// TIA Portal project "Tesis_taponado" (V20)

(* hardware
DEVICE "S7-1200 station_1"  S7-1200 Station
   slot 0: "Rack_0"  S7-1200 Rack  Rack  V1.0
   slot 1: "PLC_1"  CPU 1214C AC/DC/Rly  6ES7 214-1BG40-0XB0  V4.2
*)

// ===== PLC "PLC_1"  CPU 1214C AC/DC/Rly =====

VAR_GLOBAL   // PLC tag table "Default tag table"
   "I.G" AT %I0.1 : Bool;
   "m" AT %I0.0 : Bool;
   "final_1" AT %I0.6 : Bool;
   "Banda_1" AT %Q0.1 : Bool;
   "E0" AT %M10.0 : Bool;
   "E2" AT %M10.1 : Bool;
   "KT1" AT %M10.2 : Bool;
   "E1" AT %M10.3 : Bool;
   "Fc1" AT %M10.4 : Bool;
   "aux1" AT %M10.5 : Bool;
   "E50" AT %M10.6 : Bool;
   "E51" AT %M10.7 : Bool;
   "E52" AT %M1.0 : Bool;
   "aux2" AT %M11.1 : Bool;
   "final_2" AT %I0.7 : Bool;
   "final_3" AT %I1.0 : Bool;
   "aux3" AT %M11.2 : Bool;
   "final_4" AT %I1.1 : Bool;
   "aux4" AT %M11.3 : Bool;
   "Fc2" AT %M1.4 : Bool;
   "Fc3" AT %M1.5 : Bool;
   "Fc4" AT %M1.6 : Bool;
   "E12" AT %M1.7 : Bool;
   "E92" AT %M2.0 : Bool;
   "E11" AT %M2.1 : Bool;
   "E91" AT %M2.2 : Bool;
   "E10" AT %M2.3 : Bool;
   "E90" AT %M2.4 : Bool;
   "E20" AT %M2.5 : Bool;
   "E32" AT %M2.6 : Bool;
   "E22" AT %M2.7 : Bool;
   "KT2" AT %M3.0 : Bool;
   "E21" AT %M3.1 : Bool;
   "E31" AT %M3.2 : Bool;
   "E30" AT %M3.3 : Bool;
   "E40" AT %M3.4 : Bool;
   "E42" AT %M3.5 : Bool;
   "KT3" AT %M3.6 : Bool;
   "E41" AT %M3.7 : Bool;
   "E72" AT %M4.0 : Bool;
   "E60" AT %M4.1 : Bool;
   "E62" AT %M4.2 : Bool;
   "KT4" AT %M4.3 : Bool;
   "E61" AT %M4.4 : Bool;
   "E71" AT %M4.5 : Bool;
   "E70" AT %M4.6 : Bool;
   "Banda_2" AT %Q0.2 : Bool;
   "Banda_3" AT %Q0.3 : Bool;
   "Banda_4" AT %Q0.0 : Bool;
   "Stopped" AT %M4.7 : Bool;
   "Suspending" AT %I0.2 : Bool;
   "Aborting" AT %I0.3 : Bool;
   "aux5" AT %M5.0 : Bool;
   "UnAbort" AT %M5.1 : Bool;
   "aux6" AT %M5.2 : Bool;
   "Unsuspend" AT %M5.3 : Bool;
   "Starting" AT %M5.4 : Bool;
   "aux7" AT %M5.5 : Bool;
   "aux8" AT %M5.6 : Bool;
   "Starting_Lavado" AT %M5.7 : Bool;
   "aux9" AT %M6.0 : Bool;
   "Starting_Llenado" AT %M6.1 : Bool;
   "aux10" AT %M6.2 : Bool;
   "Starting_Taponado" AT %M6.3 : Bool;
   "aux11" AT %M6.4 : Bool;
   "Starting_Etiquetado" AT %M6.5 : Bool;
   "Start" AT %I0.4 : Bool;
   "Stop_Led" AT %Q0.5 : Bool;
   "Abort_Led" AT %Q1.0 : Bool;
   "Suspend_Led" AT %Q0.7 : Bool;
   "Start_Led" AT %Q1.1 : Bool;
   "aux12" AT %M8.7 : Bool;
END_VAR

DATA_BLOCK "DB1"   // DB1
{ S7_Optimized_Access := 'FALSE' }
VERSION : 0.1
   VAR
      UnAbort : Bool := false;
      Holding_Llenado : Bool;
      Holding_Taponado : Bool;
      Holding_Etiquetado : Bool;
      Holding_Lavado : Bool;
      Completing_Etiquetado : Bool;
      Completing_Taponado : Bool;
      Completing_Llenado : Bool;
      Completing_Lavado : Bool;
      Lavado : Bool;
      Starting : Bool;
      Starting_Lavado : Bool;
      Starting_Llenado : Bool;
      Starting_Taponado : Bool;
      Starting_Etiquetado : Bool;
      Unsuspend : Bool := false;
      Taponado : Bool;
      Etiquetado : Bool;
      Llenado : Bool;
      Aborted : Bool;
      Suspended : Bool;
      starting_plc : Bool;
      error_1 : Bool;
      error_2 : Bool;
      error_3 : Bool;
      error_4 : Bool;
   END_VAR
BEGIN
END_DATA_BLOCK

// folder: System blocks/Program resources

DATA_BLOCK "IEC_Timer_0_DB_1"   // DB2
{ S7_Optimized_Access := 'TRUE' }
AUTHOR : Simatic
FAMILY : IEC
NAME : IEC_TMR
VERSION : 1.0
// stored: InstanceOfName IEC_TIMER
"IEC_TIMER"
BEGIN
END_DATA_BLOCK

DATA_BLOCK "IEC_Timer_0_DB"   // DB3
{ S7_Optimized_Access := 'TRUE' }
AUTHOR : Simatic
FAMILY : IEC
NAME : IEC_TMR
VERSION : 1.0
// stored: InstanceOfName IEC_TIMER
"IEC_TIMER"
BEGIN
END_DATA_BLOCK

DATA_BLOCK "IEC_Timer_0_DB_2"   // DB4
{ S7_Optimized_Access := 'TRUE' }
AUTHOR : Simatic
FAMILY : IEC
NAME : IEC_TMR
VERSION : 1.0
// stored: InstanceOfName IEC_TIMER
"IEC_TIMER"
BEGIN
END_DATA_BLOCK

DATA_BLOCK "IEC_Timer_0_DB_3"   // DB5
{ S7_Optimized_Access := 'TRUE' }
AUTHOR : Simatic
FAMILY : IEC
NAME : IEC_TMR
VERSION : 1.0
// stored: InstanceOfName IEC_TIMER
"IEC_TIMER"
BEGIN
END_DATA_BLOCK

DATA_BLOCK "IEC_Timer_0_DB_4"   // DB6
{ S7_Optimized_Access := 'TRUE' }
AUTHOR : Simatic
FAMILY : IEC
NAME : IEC_TMR
VERSION : 1.0
// stored: InstanceOfName IEC_TIMER
"IEC_TIMER"
BEGIN
END_DATA_BLOCK

DATA_BLOCK "IEC_Timer_0_DB_5"   // DB7
{ S7_Optimized_Access := 'TRUE' }
AUTHOR : Simatic
FAMILY : IEC
NAME : IEC_TMR
VERSION : 1.0
// stored: InstanceOfName IEC_TIMER
"IEC_TIMER"
BEGIN
END_DATA_BLOCK

DATA_BLOCK "IEC_Timer_0_DB_6"   // DB8
{ S7_Optimized_Access := 'TRUE' }
AUTHOR : Simatic
FAMILY : IEC
NAME : IEC_TMR
VERSION : 1.0
// stored: InstanceOfName IEC_TIMER
"IEC_TIMER"
BEGIN
END_DATA_BLOCK

DATA_BLOCK "IEC_Timer_0_DB_7"   // DB9
{ S7_Optimized_Access := 'TRUE' }
AUTHOR : Simatic
FAMILY : IEC
NAME : IEC_TMR
VERSION : 1.0
// stored: InstanceOfName IEC_TIMER
"IEC_TIMER"
BEGIN
END_DATA_BLOCK

// folder: (top level)

ORGANIZATION_BLOCK "Main"   // OB1, LAD, ProgramCycle
TITLE = "Main Program Sweep (Cycle)"
{ S7_Optimized_Access := 'TRUE' }
VERSION : 0.1
   VAR_INPUT
      Initial_Call : Bool;   // Initial call of this OB
      Remanence : Bool;   // =True, if remanent data are available
   END_VAR
   VAR_TEMP
      E91 : Bool;
      np : Bool;
   END_VAR
   VAR_TEMP   // added for the SCL form of the ladder/FBD networks
      _w1 : Bool;
   END_VAR
BEGIN

REGION Network 1
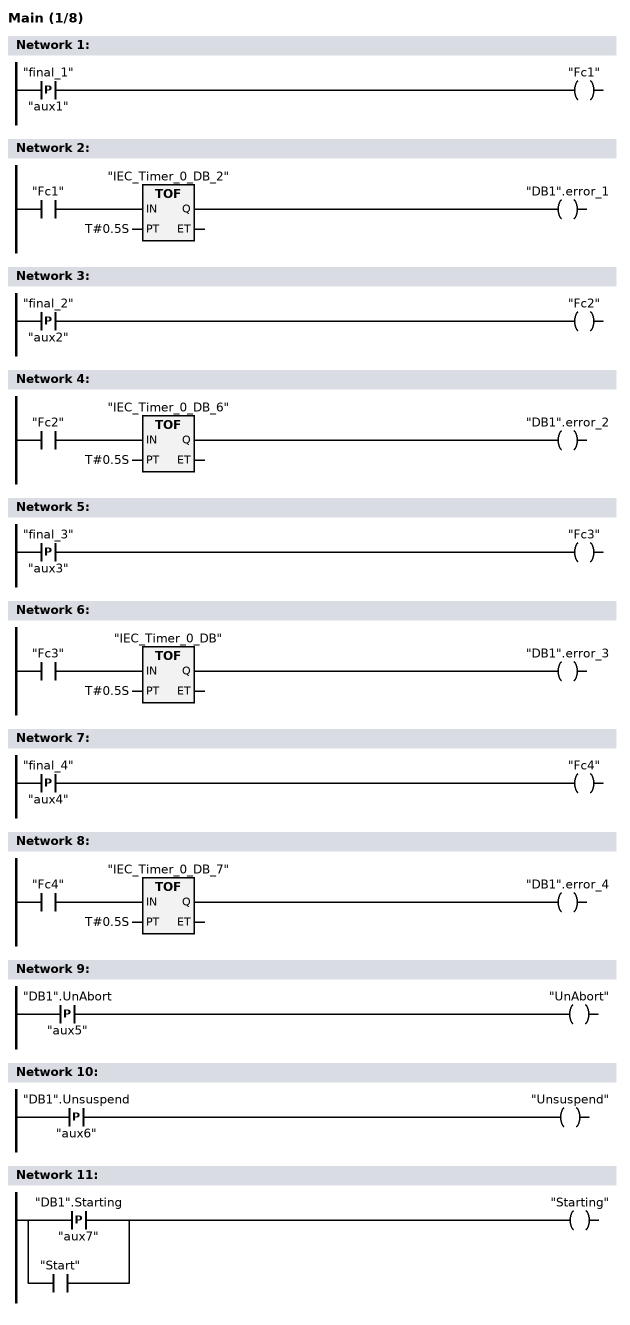
   RUNG wire#powerrail
      P_Contact(operand := "final_1", bit := "aux1")
      Coil( "Fc1" )
   END_RUNG
   // the same network as SCL:
   #_w1 := "final_1" AND NOT "aux1";   // rising edge of "final_1"
   "aux1" := "final_1";
   "Fc1" := #_w1;
END_REGION

REGION Network 2
   "IEC_Timer_0_DB_2".TOF(IN := "Fc1", PT := T#0.5S);
   "DB1".error_1 := "IEC_Timer_0_DB_2".Q;
END_REGION

REGION Network 3
   RUNG wire#powerrail
      P_Contact(operand := "final_2", bit := "aux2")
      Coil( "Fc2" )
   END_RUNG
   // the same network as SCL:
   #_w1 := "final_2" AND NOT "aux2";   // rising edge of "final_2"
   "aux2" := "final_2";
   "Fc2" := #_w1;
END_REGION

REGION Network 4
   "IEC_Timer_0_DB_6".TOF(IN := "Fc2", PT := T#0.5S);
   "DB1".error_2 := "IEC_Timer_0_DB_6".Q;
END_REGION

REGION Network 5
   RUNG wire#powerrail
      P_Contact(operand := "final_3", bit := "aux3")
      Coil( "Fc3" )
   END_RUNG
   // the same network as SCL:
   #_w1 := "final_3" AND NOT "aux3";   // rising edge of "final_3"
   "aux3" := "final_3";
   "Fc3" := #_w1;
END_REGION

REGION Network 6
   "IEC_Timer_0_DB".TOF(IN := "Fc3", PT := T#0.5S);
   "DB1".error_3 := "IEC_Timer_0_DB".Q;
END_REGION

REGION Network 7
   RUNG wire#powerrail
      P_Contact(operand := "final_4", bit := "aux4")
      Coil( "Fc4" )
   END_RUNG
   // the same network as SCL:
   #_w1 := "final_4" AND NOT "aux4";   // rising edge of "final_4"
   "aux4" := "final_4";
   "Fc4" := #_w1;
END_REGION

REGION Network 8
   "IEC_Timer_0_DB_7".TOF(IN := "Fc4", PT := T#0.5S);
   "DB1".error_4 := "IEC_Timer_0_DB_7".Q;
END_REGION

REGION Network 9
   RUNG wire#powerrail
      P_Contact(operand := "DB1".UnAbort, bit := "aux5")
      Coil( "UnAbort" )
   END_RUNG
   // the same network as SCL:
   #_w1 := "DB1".UnAbort AND NOT "aux5";   // rising edge of "DB1".UnAbort
   "aux5" := "DB1".UnAbort;
   "UnAbort" := #_w1;
END_REGION

REGION Network 10
   RUNG wire#powerrail
      P_Contact(operand := "DB1".Unsuspend, bit := "aux6")
      Coil( "Unsuspend" )
   END_RUNG
   // the same network as SCL:
   #_w1 := "DB1".Unsuspend AND NOT "aux6";   // rising edge of "DB1".Unsuspend
   "aux6" := "DB1".Unsuspend;
   "Unsuspend" := #_w1;
END_REGION

REGION Network 11
   RUNG wire#powerrail
      P_Contact(operand := "DB1".Starting, bit := "aux7")
      wire#w1
      Coil( "Starting" )
   END_RUNG
   RUNG wire#powerrail
      Contact( "Start" )
   END_RUNG wire#w1
   // the same network as SCL:
   #_w1 := "DB1".Starting AND NOT "aux7";   // rising edge of "DB1".Starting
   "aux7" := "DB1".Starting;
   "Starting" := #_w1 OR "Start";
END_REGION

REGION Network 12
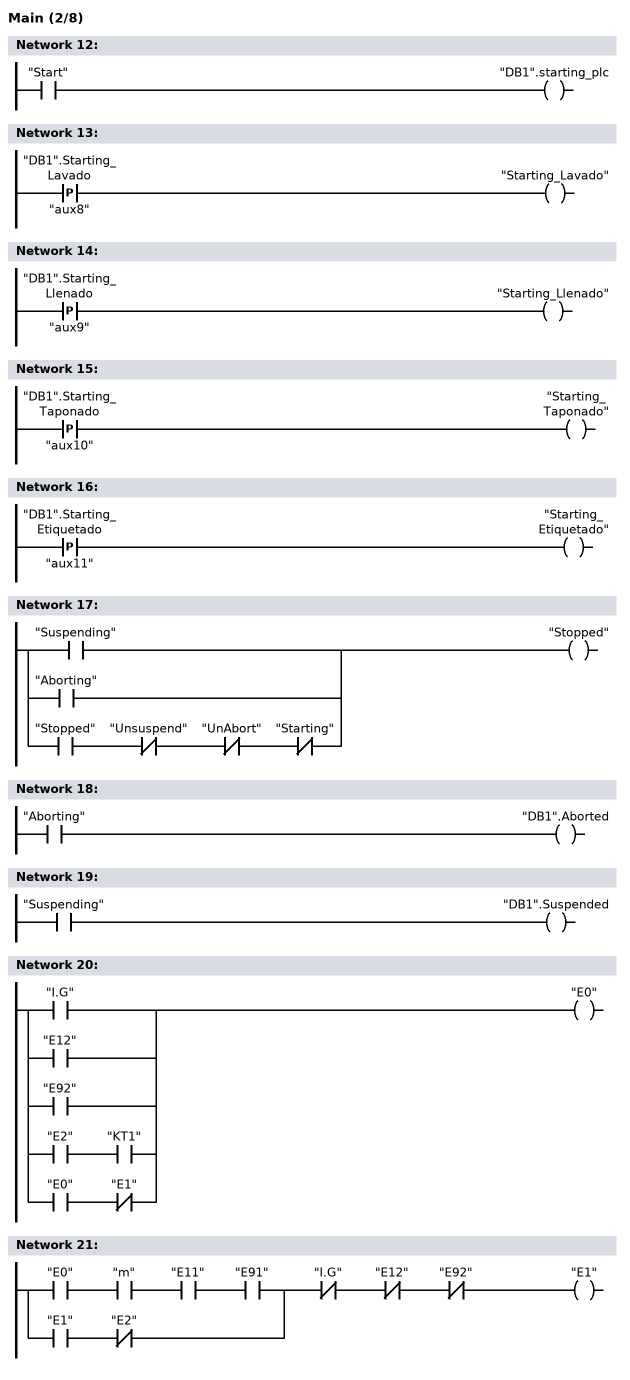
   RUNG wire#powerrail
      Contact( "Start" )
      Coil( "DB1".starting_plc )
   END_RUNG
   // the same network as SCL:
   "DB1".starting_plc := "Start";
END_REGION

REGION Network 13
   RUNG wire#powerrail
      P_Contact(operand := "DB1".Starting_Lavado, bit := "aux8")
      Coil( "Starting_Lavado" )
   END_RUNG
   // the same network as SCL:
   #_w1 := "DB1".Starting_Lavado AND NOT "aux8";   // rising edge of "DB1".Starting_Lavado
   "aux8" := "DB1".Starting_Lavado;
   "Starting_Lavado" := #_w1;
END_REGION

REGION Network 14
   RUNG wire#powerrail
      P_Contact(operand := "DB1".Starting_Llenado, bit := "aux9")
      Coil( "Starting_Llenado" )
   END_RUNG
   // the same network as SCL:
   #_w1 := "DB1".Starting_Llenado AND NOT "aux9";   // rising edge of "DB1".Starting_Llenado
   "aux9" := "DB1".Starting_Llenado;
   "Starting_Llenado" := #_w1;
END_REGION

REGION Network 15
   RUNG wire#powerrail
      P_Contact(operand := "DB1".Starting_Taponado, bit := "aux10")
      Coil( "Starting_Taponado" )
   END_RUNG
   // the same network as SCL:
   #_w1 := "DB1".Starting_Taponado AND NOT "aux10";   // rising edge of "DB1".Starting_Taponado
   "aux10" := "DB1".Starting_Taponado;
   "Starting_Taponado" := #_w1;
END_REGION

REGION Network 16
   RUNG wire#powerrail
      P_Contact(operand := "DB1".Starting_Etiquetado, bit := "aux11")
      Coil( "Starting_Etiquetado" )
   END_RUNG
   // the same network as SCL:
   #_w1 := "DB1".Starting_Etiquetado AND NOT "aux11";   // rising edge of "DB1".Starting_Etiquetado
   "aux11" := "DB1".Starting_Etiquetado;
   "Starting_Etiquetado" := #_w1;
END_REGION

REGION Network 17
   RUNG wire#powerrail
      Contact( "Suspending" )
      wire#w1
      Coil( "Stopped" )
   END_RUNG
   RUNG wire#powerrail
      Contact( "Aborting" )
   END_RUNG wire#w1
   RUNG wire#powerrail
      Contact( "Stopped" )
      I_Contact( "Unsuspend" )
      I_Contact( "UnAbort" )
      I_Contact( "Starting" )
   END_RUNG wire#w1
   // the same network as SCL:
   "Stopped" := "Suspending" OR "Aborting" OR ("Stopped" AND NOT "Unsuspend" AND NOT "UnAbort" AND NOT "Starting");
END_REGION

REGION Network 18
   RUNG wire#powerrail
      Contact( "Aborting" )
      Coil( "DB1".Aborted )
   END_RUNG
   // the same network as SCL:
   "DB1".Aborted := "Aborting";
END_REGION

REGION Network 19
   RUNG wire#powerrail
      Contact( "Suspending" )
      Coil( "DB1".Suspended )
   END_RUNG
   // the same network as SCL:
   "DB1".Suspended := "Suspending";
END_REGION

REGION Network 20
   RUNG wire#powerrail
      Contact( "I.G" )
      wire#w1
      Coil( "E0" )
   END_RUNG
   RUNG wire#powerrail
      Contact( "E12" )
   END_RUNG wire#w1
   RUNG wire#powerrail
      Contact( "E92" )
   END_RUNG wire#w1
   RUNG wire#powerrail
      Contact( "E2" )
      Contact( "KT1" )
   END_RUNG wire#w1
   RUNG wire#powerrail
      Contact( "E0" )
      I_Contact( "E1" )
   END_RUNG wire#w1
   // the same network as SCL:
   "E0" := "I.G" OR "E12" OR "E92" OR ("E2" AND "KT1") OR ("E0" AND NOT "E1");
END_REGION

REGION Network 21
   RUNG wire#powerrail
      Contact( "E0" )
      Contact( "m" )
      Contact( "E11" )
      Contact( "E91" )
      wire#w1
      I_Contact( "I.G" )
      I_Contact( "E12" )
      I_Contact( "E92" )
      Coil( "E1" )
   END_RUNG
   RUNG wire#powerrail
      Contact( "E1" )
      I_Contact( "E2" )
   END_RUNG wire#w1
   // the same network as SCL:
   "E1" := (("E0" AND "m" AND "E11" AND "E91") OR ("E1" AND NOT "E2")) AND NOT "I.G" AND NOT "E12" AND NOT "E92";
END_REGION

REGION Network 22
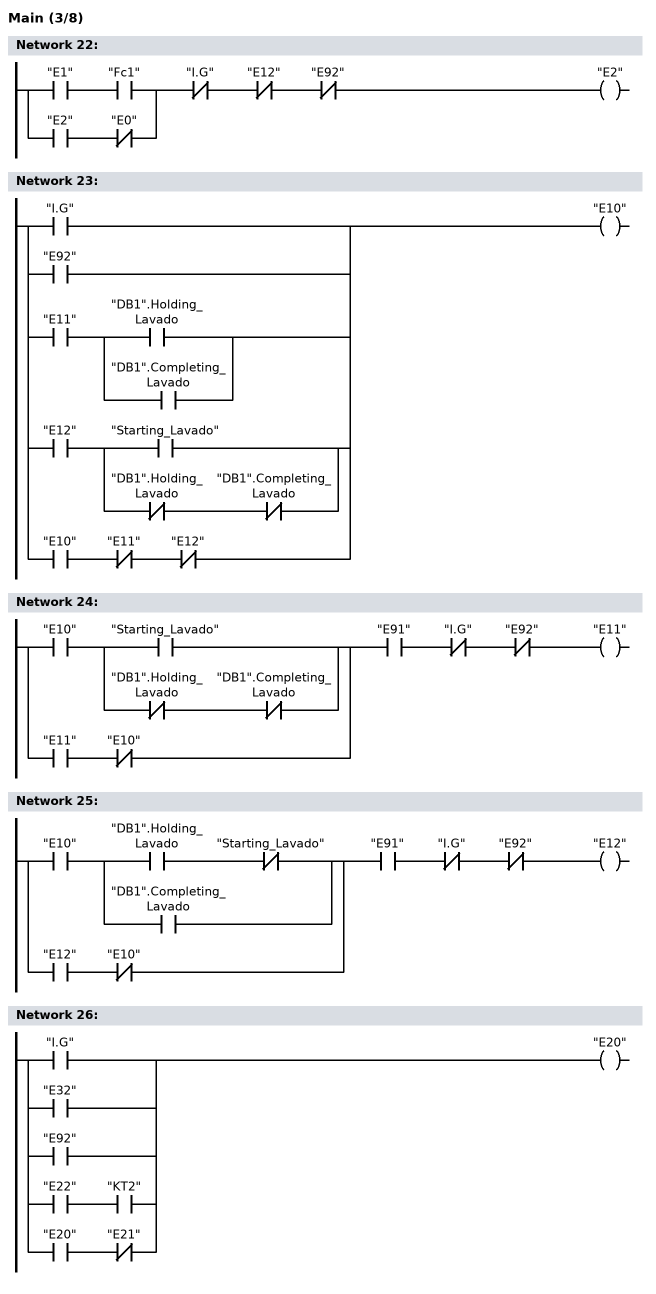
   RUNG wire#powerrail
      Contact( "E1" )
      Contact( "Fc1" )
      wire#w1
      I_Contact( "I.G" )
      I_Contact( "E12" )
      I_Contact( "E92" )
      Coil( "E2" )
   END_RUNG
   RUNG wire#powerrail
      Contact( "E2" )
      I_Contact( "E0" )
   END_RUNG wire#w1
   // the same network as SCL:
   "E2" := (("E1" AND "Fc1") OR ("E2" AND NOT "E0")) AND NOT "I.G" AND NOT "E12" AND NOT "E92";
END_REGION

REGION Network 23
   RUNG wire#powerrail
      Contact( "I.G" )
      wire#w1
      Coil( "E10" )
   END_RUNG
   RUNG wire#powerrail
      Contact( "E92" )
   END_RUNG wire#w1
   RUNG wire#powerrail
      Contact( "E11" )
      wire#w2
      Contact( "DB1".Holding_Lavado )
   END_RUNG wire#w1
   RUNG wire#w2
      Contact( "DB1".Completing_Lavado )
   END_RUNG wire#w1
   RUNG wire#powerrail
      Contact( "E12" )
      wire#w3
      Contact( "Starting_Lavado" )
   END_RUNG wire#w1
   RUNG wire#w3
      I_Contact( "DB1".Holding_Lavado )
      I_Contact( "DB1".Completing_Lavado )
   END_RUNG wire#w1
   RUNG wire#powerrail
      Contact( "E10" )
      I_Contact( "E11" )
      I_Contact( "E12" )
   END_RUNG wire#w1
   // the same network as SCL:
   "E10" := "I.G" OR "E92" OR ("E11" AND ("DB1".Holding_Lavado OR "DB1".Completing_Lavado)) OR ("E12" AND ("Starting_Lavado" OR (NOT "DB1".Holding_Lavado AND NOT "DB1".Completing_Lavado))) OR ("E10" AND NOT "E11" AND NOT "E12");
END_REGION

REGION Network 24
   RUNG wire#powerrail
      Contact( "E10" )
      wire#w1
      Contact( "Starting_Lavado" )
      wire#w2
      Contact( "E91" )
      I_Contact( "I.G" )
      I_Contact( "E92" )
      Coil( "E11" )
   END_RUNG
   RUNG wire#w1
      I_Contact( "DB1".Holding_Lavado )
      I_Contact( "DB1".Completing_Lavado )
   END_RUNG wire#w2
   RUNG wire#powerrail
      Contact( "E11" )
      I_Contact( "E10" )
   END_RUNG wire#w2
   // the same network as SCL:
   "E11" := (("E10" AND ("Starting_Lavado" OR (NOT "DB1".Holding_Lavado AND NOT "DB1".Completing_Lavado))) OR ("E11" AND NOT "E10")) AND "E91" AND NOT "I.G" AND NOT "E92";
END_REGION

REGION Network 25
   RUNG wire#powerrail
      Contact( "E10" )
      wire#w1
      Contact( "DB1".Holding_Lavado )
      I_Contact( "Starting_Lavado" )
      wire#w2
      Contact( "E91" )
      I_Contact( "I.G" )
      I_Contact( "E92" )
      Coil( "E12" )
   END_RUNG
   RUNG wire#w1
      Contact( "DB1".Completing_Lavado )
   END_RUNG wire#w2
   RUNG wire#powerrail
      Contact( "E12" )
      I_Contact( "E10" )
   END_RUNG wire#w2
   // the same network as SCL:
   "E12" := (("E10" AND (("DB1".Holding_Lavado AND NOT "Starting_Lavado") OR "DB1".Completing_Lavado)) OR ("E12" AND NOT "E10")) AND "E91" AND NOT "I.G" AND NOT "E92";
END_REGION

REGION Network 26
   RUNG wire#powerrail
      Contact( "I.G" )
      wire#w1
      Coil( "E20" )
   END_RUNG
   RUNG wire#powerrail
      Contact( "E32" )
   END_RUNG wire#w1
   RUNG wire#powerrail
      Contact( "E92" )
   END_RUNG wire#w1
   RUNG wire#powerrail
      Contact( "E22" )
      Contact( "KT2" )
   END_RUNG wire#w1
   RUNG wire#powerrail
      Contact( "E20" )
      I_Contact( "E21" )
   END_RUNG wire#w1
   // the same network as SCL:
   "E20" := "I.G" OR "E32" OR "E92" OR ("E22" AND "KT2") OR ("E20" AND NOT "E21");
END_REGION

REGION Network 27
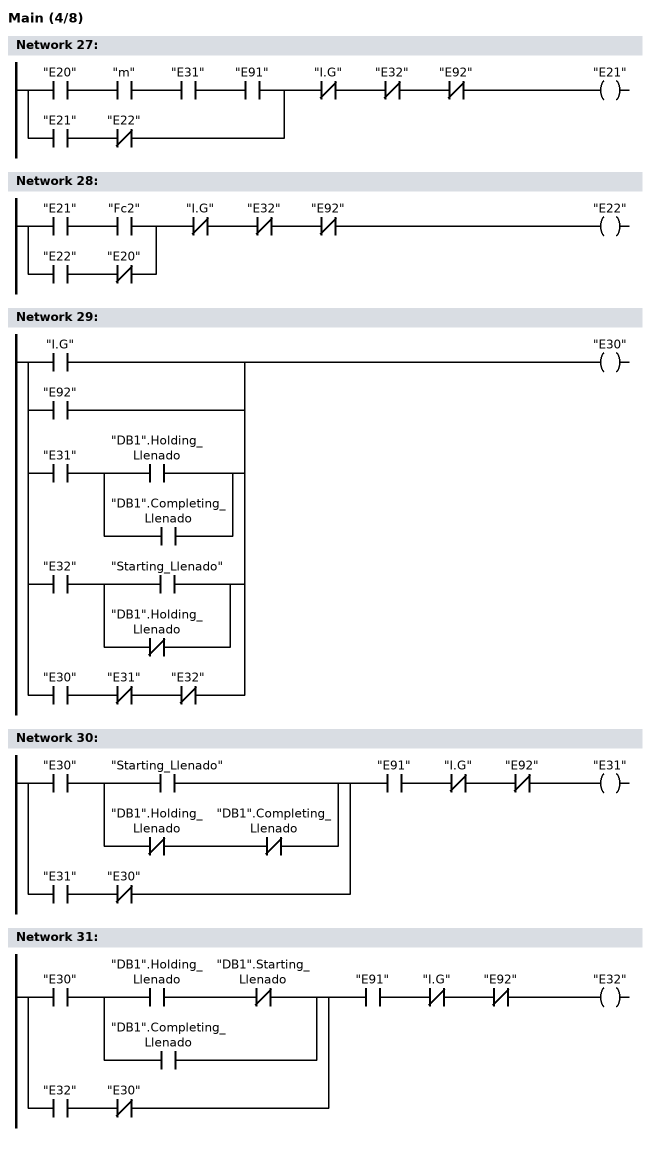
   RUNG wire#powerrail
      Contact( "E20" )
      Contact( "m" )
      Contact( "E31" )
      Contact( "E91" )
      wire#w1
      I_Contact( "I.G" )
      I_Contact( "E32" )
      I_Contact( "E92" )
      Coil( "E21" )
   END_RUNG
   RUNG wire#powerrail
      Contact( "E21" )
      I_Contact( "E22" )
   END_RUNG wire#w1
   // the same network as SCL:
   "E21" := (("E20" AND "m" AND "E31" AND "E91") OR ("E21" AND NOT "E22")) AND NOT "I.G" AND NOT "E32" AND NOT "E92";
END_REGION

REGION Network 28
   RUNG wire#powerrail
      Contact( "E21" )
      Contact( "Fc2" )
      wire#w1
      I_Contact( "I.G" )
      I_Contact( "E32" )
      I_Contact( "E92" )
      Coil( "E22" )
   END_RUNG
   RUNG wire#powerrail
      Contact( "E22" )
      I_Contact( "E20" )
   END_RUNG wire#w1
   // the same network as SCL:
   "E22" := (("E21" AND "Fc2") OR ("E22" AND NOT "E20")) AND NOT "I.G" AND NOT "E32" AND NOT "E92";
END_REGION

REGION Network 29
   RUNG wire#powerrail
      Contact( "I.G" )
      wire#w1
      Coil( "E30" )
   END_RUNG
   RUNG wire#powerrail
      Contact( "E92" )
   END_RUNG wire#w1
   RUNG wire#powerrail
      Contact( "E31" )
      wire#w2
      Contact( "DB1".Holding_Llenado )
   END_RUNG wire#w1
   RUNG wire#w2
      Contact( "DB1".Completing_Llenado )
   END_RUNG wire#w1
   RUNG wire#powerrail
      Contact( "E32" )
      wire#w3
      Contact( "Starting_Llenado" )
   END_RUNG wire#w1
   RUNG wire#w3
      I_Contact( "DB1".Holding_Llenado )
   END_RUNG wire#w1
   RUNG wire#powerrail
      Contact( "E30" )
      I_Contact( "E31" )
      I_Contact( "E32" )
   END_RUNG wire#w1
   // the same network as SCL:
   "E30" := "I.G" OR "E92" OR ("E31" AND ("DB1".Holding_Llenado OR "DB1".Completing_Llenado)) OR ("E32" AND ("Starting_Llenado" OR NOT "DB1".Holding_Llenado)) OR ("E30" AND NOT "E31" AND NOT "E32");
END_REGION

REGION Network 30
   RUNG wire#powerrail
      Contact( "E30" )
      wire#w1
      Contact( "Starting_Llenado" )
      wire#w2
      Contact( "E91" )
      I_Contact( "I.G" )
      I_Contact( "E92" )
      Coil( "E31" )
   END_RUNG
   RUNG wire#w1
      I_Contact( "DB1".Holding_Llenado )
      I_Contact( "DB1".Completing_Llenado )
   END_RUNG wire#w2
   RUNG wire#powerrail
      Contact( "E31" )
      I_Contact( "E30" )
   END_RUNG wire#w2
   // the same network as SCL:
   "E31" := (("E30" AND ("Starting_Llenado" OR (NOT "DB1".Holding_Llenado AND NOT "DB1".Completing_Llenado))) OR ("E31" AND NOT "E30")) AND "E91" AND NOT "I.G" AND NOT "E92";
END_REGION

REGION Network 31
   RUNG wire#powerrail
      Contact( "E30" )
      wire#w1
      Contact( "DB1".Holding_Llenado )
      I_Contact( "DB1".Starting_Llenado )
      wire#w2
      Contact( "E91" )
      I_Contact( "I.G" )
      I_Contact( "E92" )
      Coil( "E32" )
   END_RUNG
   RUNG wire#w1
      Contact( "DB1".Completing_Llenado )
   END_RUNG wire#w2
   RUNG wire#powerrail
      Contact( "E32" )
      I_Contact( "E30" )
   END_RUNG wire#w2
   // the same network as SCL:
   "E32" := (("E30" AND (("DB1".Holding_Llenado AND NOT "DB1".Starting_Llenado) OR "DB1".Completing_Llenado)) OR ("E32" AND NOT "E30")) AND "E91" AND NOT "I.G" AND NOT "E92";
END_REGION

REGION Network 32
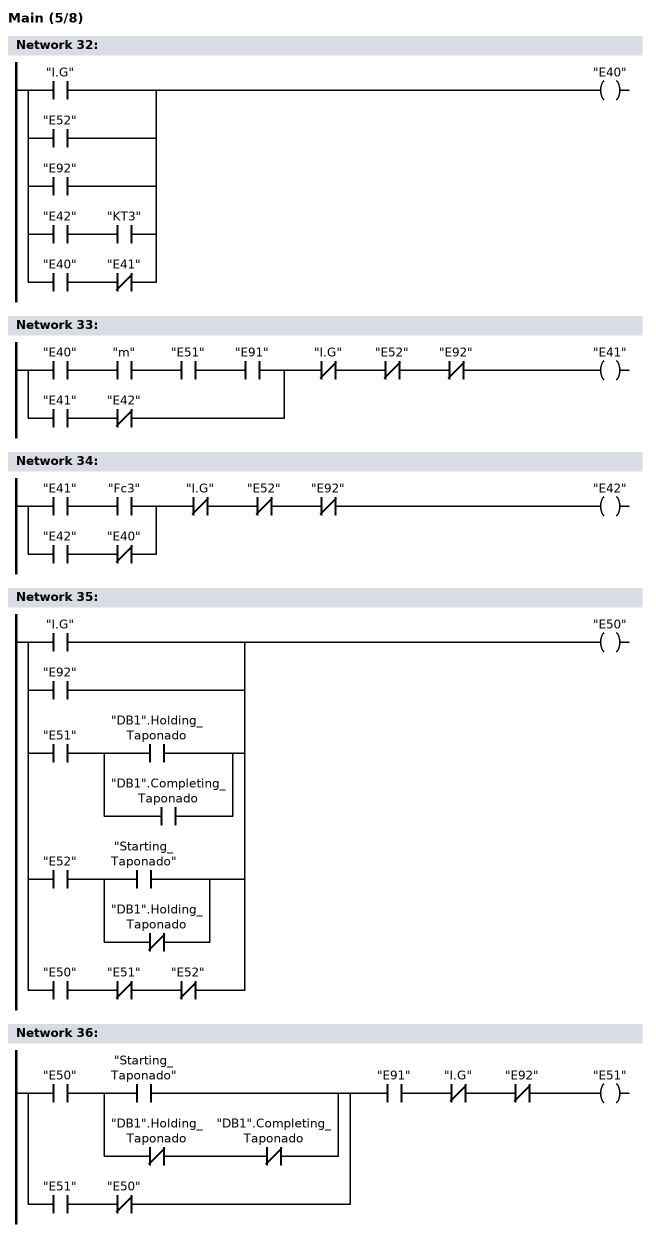
   RUNG wire#powerrail
      Contact( "I.G" )
      wire#w1
      Coil( "E40" )
   END_RUNG
   RUNG wire#powerrail
      Contact( "E52" )
   END_RUNG wire#w1
   RUNG wire#powerrail
      Contact( "E92" )
   END_RUNG wire#w1
   RUNG wire#powerrail
      Contact( "E42" )
      Contact( "KT3" )
   END_RUNG wire#w1
   RUNG wire#powerrail
      Contact( "E40" )
      I_Contact( "E41" )
   END_RUNG wire#w1
   // the same network as SCL:
   "E40" := "I.G" OR "E52" OR "E92" OR ("E42" AND "KT3") OR ("E40" AND NOT "E41");
END_REGION

REGION Network 33
   RUNG wire#powerrail
      Contact( "E40" )
      Contact( "m" )
      Contact( "E51" )
      Contact( "E91" )
      wire#w1
      I_Contact( "I.G" )
      I_Contact( "E52" )
      I_Contact( "E92" )
      Coil( "E41" )
   END_RUNG
   RUNG wire#powerrail
      Contact( "E41" )
      I_Contact( "E42" )
   END_RUNG wire#w1
   // the same network as SCL:
   "E41" := (("E40" AND "m" AND "E51" AND "E91") OR ("E41" AND NOT "E42")) AND NOT "I.G" AND NOT "E52" AND NOT "E92";
END_REGION

REGION Network 34
   RUNG wire#powerrail
      Contact( "E41" )
      Contact( "Fc3" )
      wire#w1
      I_Contact( "I.G" )
      I_Contact( "E52" )
      I_Contact( "E92" )
      Coil( "E42" )
   END_RUNG
   RUNG wire#powerrail
      Contact( "E42" )
      I_Contact( "E40" )
   END_RUNG wire#w1
   // the same network as SCL:
   "E42" := (("E41" AND "Fc3") OR ("E42" AND NOT "E40")) AND NOT "I.G" AND NOT "E52" AND NOT "E92";
END_REGION

REGION Network 35
   RUNG wire#powerrail
      Contact( "I.G" )
      wire#w1
      Coil( "E50" )
   END_RUNG
   RUNG wire#powerrail
      Contact( "E92" )
   END_RUNG wire#w1
   RUNG wire#powerrail
      Contact( "E51" )
      wire#w2
      Contact( "DB1".Holding_Taponado )
   END_RUNG wire#w1
   RUNG wire#w2
      Contact( "DB1".Completing_Taponado )
   END_RUNG wire#w1
   RUNG wire#powerrail
      Contact( "E52" )
      wire#w3
      Contact( "Starting_Taponado" )
   END_RUNG wire#w1
   RUNG wire#w3
      I_Contact( "DB1".Holding_Taponado )
   END_RUNG wire#w1
   RUNG wire#powerrail
      Contact( "E50" )
      I_Contact( "E51" )
      I_Contact( "E52" )
   END_RUNG wire#w1
   // the same network as SCL:
   "E50" := "I.G" OR "E92" OR ("E51" AND ("DB1".Holding_Taponado OR "DB1".Completing_Taponado)) OR ("E52" AND ("Starting_Taponado" OR NOT "DB1".Holding_Taponado)) OR ("E50" AND NOT "E51" AND NOT "E52");
END_REGION

REGION Network 36
   RUNG wire#powerrail
      Contact( "E50" )
      wire#w1
      Contact( "Starting_Taponado" )
      wire#w2
      Contact( "E91" )
      I_Contact( "I.G" )
      I_Contact( "E92" )
      Coil( "E51" )
   END_RUNG
   RUNG wire#w1
      I_Contact( "DB1".Holding_Taponado )
      I_Contact( "DB1".Completing_Taponado )
   END_RUNG wire#w2
   RUNG wire#powerrail
      Contact( "E51" )
      I_Contact( "E50" )
   END_RUNG wire#w2
   // the same network as SCL:
   "E51" := (("E50" AND ("Starting_Taponado" OR (NOT "DB1".Holding_Taponado AND NOT "DB1".Completing_Taponado))) OR ("E51" AND NOT "E50")) AND "E91" AND NOT "I.G" AND NOT "E92";
END_REGION

REGION Network 37
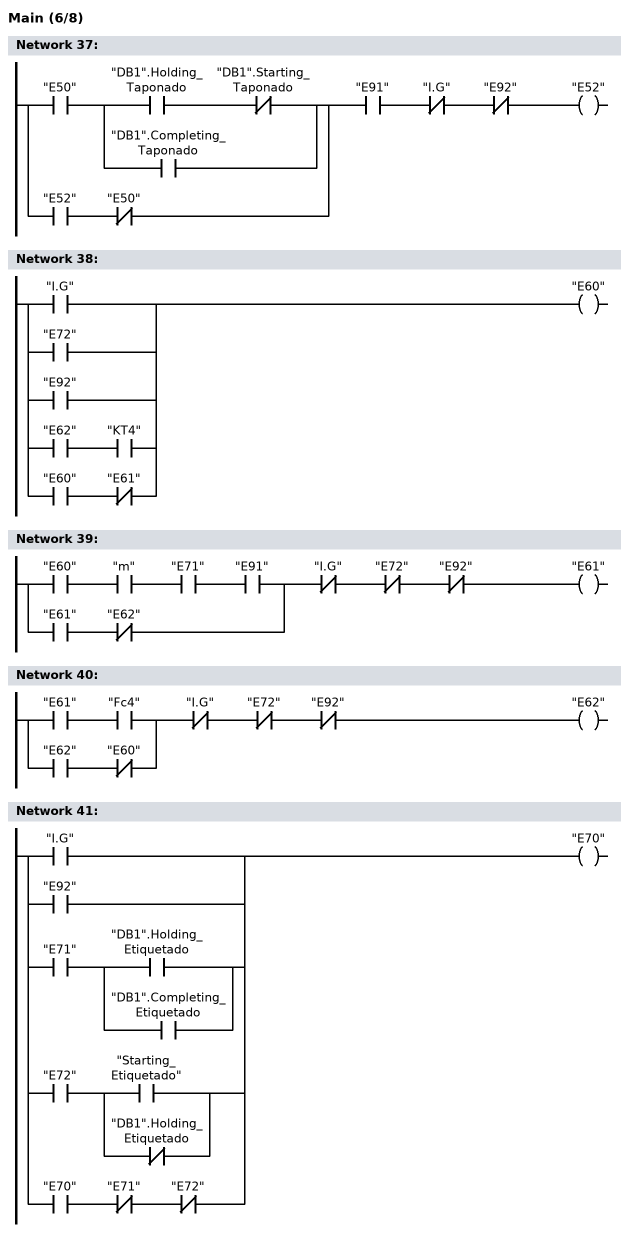
   RUNG wire#powerrail
      Contact( "E50" )
      wire#w1
      Contact( "DB1".Holding_Taponado )
      I_Contact( "DB1".Starting_Taponado )
      wire#w2
      Contact( "E91" )
      I_Contact( "I.G" )
      I_Contact( "E92" )
      Coil( "E52" )
   END_RUNG
   RUNG wire#w1
      Contact( "DB1".Completing_Taponado )
   END_RUNG wire#w2
   RUNG wire#powerrail
      Contact( "E52" )
      I_Contact( "E50" )
   END_RUNG wire#w2
   // the same network as SCL:
   "E52" := (("E50" AND (("DB1".Holding_Taponado AND NOT "DB1".Starting_Taponado) OR "DB1".Completing_Taponado)) OR ("E52" AND NOT "E50")) AND "E91" AND NOT "I.G" AND NOT "E92";
END_REGION

REGION Network 38
   RUNG wire#powerrail
      Contact( "I.G" )
      wire#w1
      Coil( "E60" )
   END_RUNG
   RUNG wire#powerrail
      Contact( "E72" )
   END_RUNG wire#w1
   RUNG wire#powerrail
      Contact( "E92" )
   END_RUNG wire#w1
   RUNG wire#powerrail
      Contact( "E62" )
      Contact( "KT4" )
   END_RUNG wire#w1
   RUNG wire#powerrail
      Contact( "E60" )
      I_Contact( "E61" )
   END_RUNG wire#w1
   // the same network as SCL:
   "E60" := "I.G" OR "E72" OR "E92" OR ("E62" AND "KT4") OR ("E60" AND NOT "E61");
END_REGION

REGION Network 39
   RUNG wire#powerrail
      Contact( "E60" )
      Contact( "m" )
      Contact( "E71" )
      Contact( "E91" )
      wire#w1
      I_Contact( "I.G" )
      I_Contact( "E72" )
      I_Contact( "E92" )
      Coil( "E61" )
   END_RUNG
   RUNG wire#powerrail
      Contact( "E61" )
      I_Contact( "E62" )
   END_RUNG wire#w1
   // the same network as SCL:
   "E61" := (("E60" AND "m" AND "E71" AND "E91") OR ("E61" AND NOT "E62")) AND NOT "I.G" AND NOT "E72" AND NOT "E92";
END_REGION

REGION Network 40
   RUNG wire#powerrail
      Contact( "E61" )
      Contact( "Fc4" )
      wire#w1
      I_Contact( "I.G" )
      I_Contact( "E72" )
      I_Contact( "E92" )
      Coil( "E62" )
   END_RUNG
   RUNG wire#powerrail
      Contact( "E62" )
      I_Contact( "E60" )
   END_RUNG wire#w1
   // the same network as SCL:
   "E62" := (("E61" AND "Fc4") OR ("E62" AND NOT "E60")) AND NOT "I.G" AND NOT "E72" AND NOT "E92";
END_REGION

REGION Network 41
   RUNG wire#powerrail
      Contact( "I.G" )
      wire#w1
      Coil( "E70" )
   END_RUNG
   RUNG wire#powerrail
      Contact( "E92" )
   END_RUNG wire#w1
   RUNG wire#powerrail
      Contact( "E71" )
      wire#w2
      Contact( "DB1".Holding_Etiquetado )
   END_RUNG wire#w1
   RUNG wire#w2
      Contact( "DB1".Completing_Etiquetado )
   END_RUNG wire#w1
   RUNG wire#powerrail
      Contact( "E72" )
      wire#w3
      Contact( "Starting_Etiquetado" )
   END_RUNG wire#w1
   RUNG wire#w3
      I_Contact( "DB1".Holding_Etiquetado )
   END_RUNG wire#w1
   RUNG wire#powerrail
      Contact( "E70" )
      I_Contact( "E71" )
      I_Contact( "E72" )
   END_RUNG wire#w1
   // the same network as SCL:
   "E70" := "I.G" OR "E92" OR ("E71" AND ("DB1".Holding_Etiquetado OR "DB1".Completing_Etiquetado)) OR ("E72" AND ("Starting_Etiquetado" OR NOT "DB1".Holding_Etiquetado)) OR ("E70" AND NOT "E71" AND NOT "E72");
END_REGION

REGION Network 42
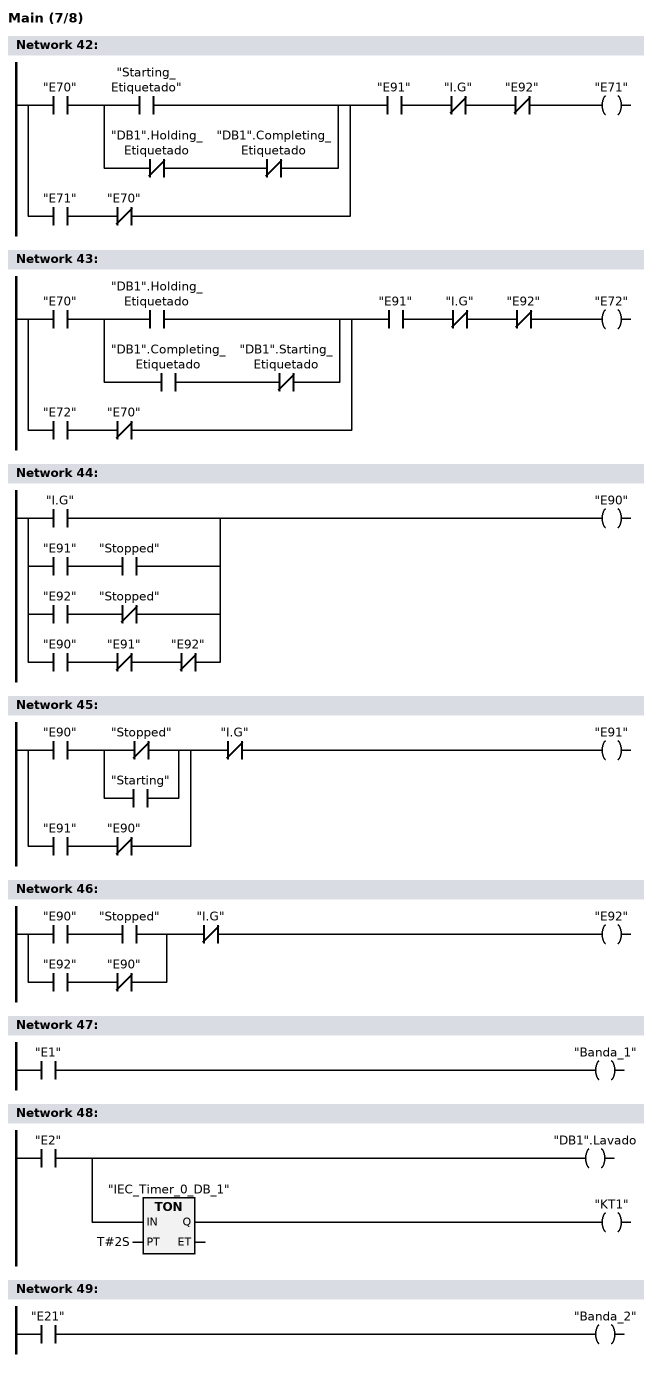
   RUNG wire#powerrail
      Contact( "E70" )
      wire#w1
      Contact( "Starting_Etiquetado" )
      wire#w2
      Contact( "E91" )
      I_Contact( "I.G" )
      I_Contact( "E92" )
      Coil( "E71" )
   END_RUNG
   RUNG wire#w1
      I_Contact( "DB1".Holding_Etiquetado )
      I_Contact( "DB1".Completing_Etiquetado )
   END_RUNG wire#w2
   RUNG wire#powerrail
      Contact( "E71" )
      I_Contact( "E70" )
   END_RUNG wire#w2
   // the same network as SCL:
   "E71" := (("E70" AND ("Starting_Etiquetado" OR (NOT "DB1".Holding_Etiquetado AND NOT "DB1".Completing_Etiquetado))) OR ("E71" AND NOT "E70")) AND "E91" AND NOT "I.G" AND NOT "E92";
END_REGION

REGION Network 43
   RUNG wire#powerrail
      Contact( "E70" )
      wire#w1
      Contact( "DB1".Holding_Etiquetado )
      wire#w2
      Contact( "E91" )
      I_Contact( "I.G" )
      I_Contact( "E92" )
      Coil( "E72" )
   END_RUNG
   RUNG wire#w1
      Contact( "DB1".Completing_Etiquetado )
      I_Contact( "DB1".Starting_Etiquetado )
   END_RUNG wire#w2
   RUNG wire#powerrail
      Contact( "E72" )
      I_Contact( "E70" )
   END_RUNG wire#w2
   // the same network as SCL:
   "E72" := (("E70" AND ("DB1".Holding_Etiquetado OR ("DB1".Completing_Etiquetado AND NOT "DB1".Starting_Etiquetado))) OR ("E72" AND NOT "E70")) AND "E91" AND NOT "I.G" AND NOT "E92";
END_REGION

REGION Network 44
   RUNG wire#powerrail
      Contact( "I.G" )
      wire#w1
      Coil( "E90" )
   END_RUNG
   RUNG wire#powerrail
      Contact( "E91" )
      Contact( "Stopped" )
   END_RUNG wire#w1
   RUNG wire#powerrail
      Contact( "E92" )
      I_Contact( "Stopped" )
   END_RUNG wire#w1
   RUNG wire#powerrail
      Contact( "E90" )
      I_Contact( "E91" )
      I_Contact( "E92" )
   END_RUNG wire#w1
   // the same network as SCL:
   "E90" := "I.G" OR ("E91" AND "Stopped") OR ("E92" AND NOT "Stopped") OR ("E90" AND NOT "E91" AND NOT "E92");
END_REGION

REGION Network 45
   RUNG wire#powerrail
      Contact( "E90" )
      wire#w1
      I_Contact( "Stopped" )
      wire#w2
      I_Contact( "I.G" )
      Coil( "E91" )
   END_RUNG
   RUNG wire#w1
      Contact( "Starting" )
   END_RUNG wire#w2
   RUNG wire#powerrail
      Contact( "E91" )
      I_Contact( "E90" )
   END_RUNG wire#w2
   // the same network as SCL:
   "E91" := (("E90" AND (NOT "Stopped" OR "Starting")) OR ("E91" AND NOT "E90")) AND NOT "I.G";
END_REGION

REGION Network 46
   RUNG wire#powerrail
      Contact( "E90" )
      Contact( "Stopped" )
      wire#w1
      I_Contact( "I.G" )
      Coil( "E92" )
   END_RUNG
   RUNG wire#powerrail
      Contact( "E92" )
      I_Contact( "E90" )
   END_RUNG wire#w1
   // the same network as SCL:
   "E92" := (("E90" AND "Stopped") OR ("E92" AND NOT "E90")) AND NOT "I.G";
END_REGION

REGION Network 47
   RUNG wire#powerrail
      Contact( "E1" )
      Coil( "Banda_1" )
   END_RUNG
   // the same network as SCL:
   "Banda_1" := "E1";
END_REGION

REGION Network 48
   "DB1".Lavado := "E2";
   "IEC_Timer_0_DB_1".TON(IN := "E2", PT := T#2S);
   "KT1" := "IEC_Timer_0_DB_1".Q;
END_REGION

REGION Network 49
   RUNG wire#powerrail
      Contact( "E21" )
      Coil( "Banda_2" )
   END_RUNG
   // the same network as SCL:
   "Banda_2" := "E21";
END_REGION

REGION Network 50
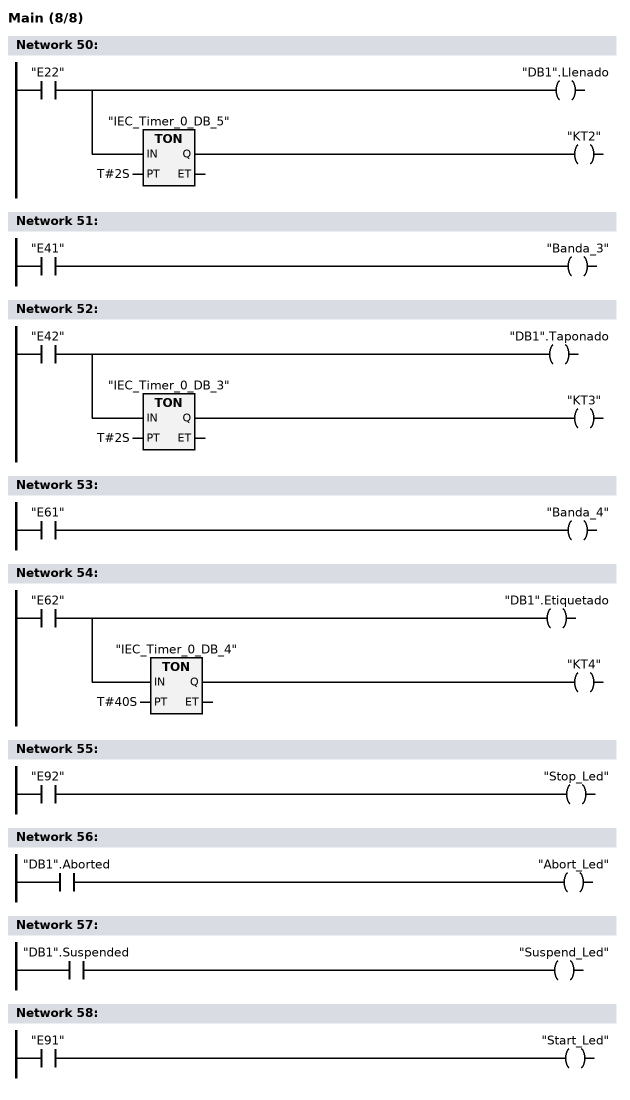
   "DB1".Llenado := "E22";
   "IEC_Timer_0_DB_5".TON(IN := "E22", PT := T#2S);
   "KT2" := "IEC_Timer_0_DB_5".Q;
END_REGION

REGION Network 51
   RUNG wire#powerrail
      Contact( "E41" )
      Coil( "Banda_3" )
   END_RUNG
   // the same network as SCL:
   "Banda_3" := "E41";
END_REGION

REGION Network 52
   "DB1".Taponado := "E42";
   "IEC_Timer_0_DB_3".TON(IN := "E42", PT := T#2S);
   "KT3" := "IEC_Timer_0_DB_3".Q;
END_REGION

REGION Network 53
   RUNG wire#powerrail
      Contact( "E61" )
      Coil( "Banda_4" )
   END_RUNG
   // the same network as SCL:
   "Banda_4" := "E61";
END_REGION

REGION Network 54
   "DB1".Etiquetado := "E62";
   "IEC_Timer_0_DB_4".TON(IN := "E62", PT := T#40S);
   "KT4" := "IEC_Timer_0_DB_4".Q;
END_REGION

REGION Network 55
   RUNG wire#powerrail
      Contact( "E92" )
      Coil( "Stop_Led" )
   END_RUNG
   // the same network as SCL:
   "Stop_Led" := "E92";
END_REGION

REGION Network 56
   RUNG wire#powerrail
      Contact( "DB1".Aborted )
      Coil( "Abort_Led" )
   END_RUNG
   // the same network as SCL:
   "Abort_Led" := "DB1".Aborted;
END_REGION

REGION Network 57
   RUNG wire#powerrail
      Contact( "DB1".Suspended )
      Coil( "Suspend_Led" )
   END_RUNG
   // the same network as SCL:
   "Suspend_Led" := "DB1".Suspended;
END_REGION

REGION Network 58
   RUNG wire#powerrail
      Contact( "E91" )
      Coil( "Start_Led" )
   END_RUNG
   // the same network as SCL:
   "Start_Led" := "E91";
END_REGION
END_ORGANIZATION_BLOCK